FUNCTION_BLOCK Payload_B IMPLEMENTS I_Payload_B
VAR_INPUT
END_VAR
VAR_OUTPUT
END_VAR
VAR
	bPayload : BOOL;
END_VAR

END_FUNCTION_BLOCK

(* stored: Version 1.1.0.1, ProductVersion 3.1.4024.2
   POU Payload_B: Id {8ddd06a1-3223-421e-855f-9bd61f22ab00}, SpecialFunc None *)
